// ==============================================================================
// DB_Mechs - РњР°СЃРёРІРё РјРµС…Р°РЅС–Р·РјС–РІ
// ==============================================================================
// Project  : Elevator_System
// Author   : Engineering Team
// Version  : 2.0.0
// Generated: 2026-03-20 10:46:50
// ==============================================================================

DATA_BLOCK "DB_Mechs"
{ S7_Optimized_Access := 'TRUE' }
VERSION : 1.0

VAR
    // ===================================================================
    // Р‘Р°Р·РѕРІР° С€РёРЅР° РјРµС…Р°РЅС–Р·РјС–РІ (СѓСЃС– СЃР»РѕС‚Рё 0..255)
    // ===================================================================
    Mechs : ARRAY [0..255] OF "UDT_BaseMechanism";

    // Р РµРґР»РµСЂРё: 2 С€С‚, РјР°СЃРёРІ [0..1]
    Redler : ARRAY [0..1] OF "UDT_Redler";

    // РќРѕСЂС–С—: 2 С€С‚, РјР°СЃРёРІ [0..1]
    Noria : ARRAY [0..1] OF "UDT_Noria";

    // Р—Р°СЃСѓРІРєРё: 2 С€С‚, РјР°СЃРёРІ [0..1]
    Gate : ARRAY [0..1] OF "UDT_Gate2P";

    // Р’РµРЅС‚РёР»СЏС‚РѕСЂРё: 1 С€С‚, РјР°СЃРёРІ [0..0]
    Fan : ARRAY [0..0] OF "UDT_Fan";

END_VAR

BEGIN
END_DATA_BLOCK
